TYPE POZICIJA :
STRUCT
	A: INT;
	Y: INT;
	Z: INT;
	P: INT;
END_STRUCT
END_TYPE

(* stored: Version 1.1.0.1, ProductVersion 3.1.4024.12
   DUT POZICIJA: Id {4e000258-6df1-4ac0-ac7b-1648fb7ac8d9} *)
